TYPE size_t : DWORD; END_TYPE

(* stored: Version 1.1.0.1
   DUT size_t: Id {996bedc0-9977-4b0b-b46f-6d7f32597d03} *)
